// Mitsubishi GX Works2 project: Ex3   PLC: Q03UDV

PROGRAM MAIN
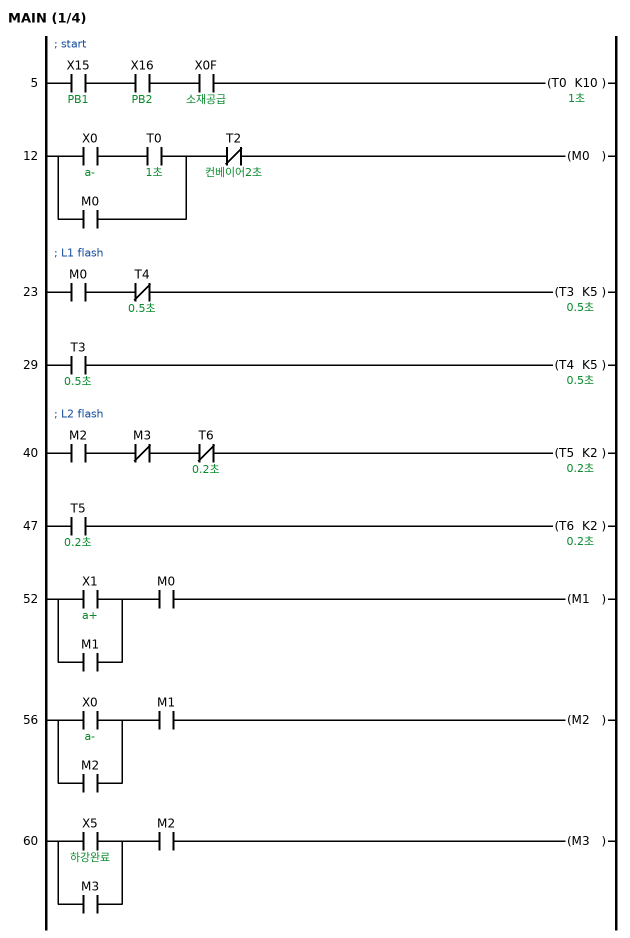
; start
5     LD      X15  ; PB1
      AND     X16  ; PB2
      AND     X0F  ; 소재공급
      OUT     T0 K10  ; 1초
12    LD      X0  ; a-
      AND     T0  ; 1초
      OR      M0
      ANI     T2  ; 컨베이어2초
      OUT     M0
; L1 flash
23    LD      M0
      ANI     T4  ; 0.5초
      OUT     T3 K5  ; 0.5초
29    LD      T3  ; 0.5초
      OUT     T4 K5  ; 0.5초
; L2 flash
40    LD      M2
      ANI     M3
      ANI     T6  ; 0.2초
      OUT     T5 K2  ; 0.2초
47    LD      T5  ; 0.2초
      OUT     T6 K2  ; 0.2초
52    LD      X1  ; a+
      OR      M1
      AND     M0
      OUT     M1
56    LD      X0  ; a-
      OR      M2
      AND     M1
      OUT     M2
60    LD      X5  ; 하강완료
      OR      M3
      AND     M2
      OUT     M3
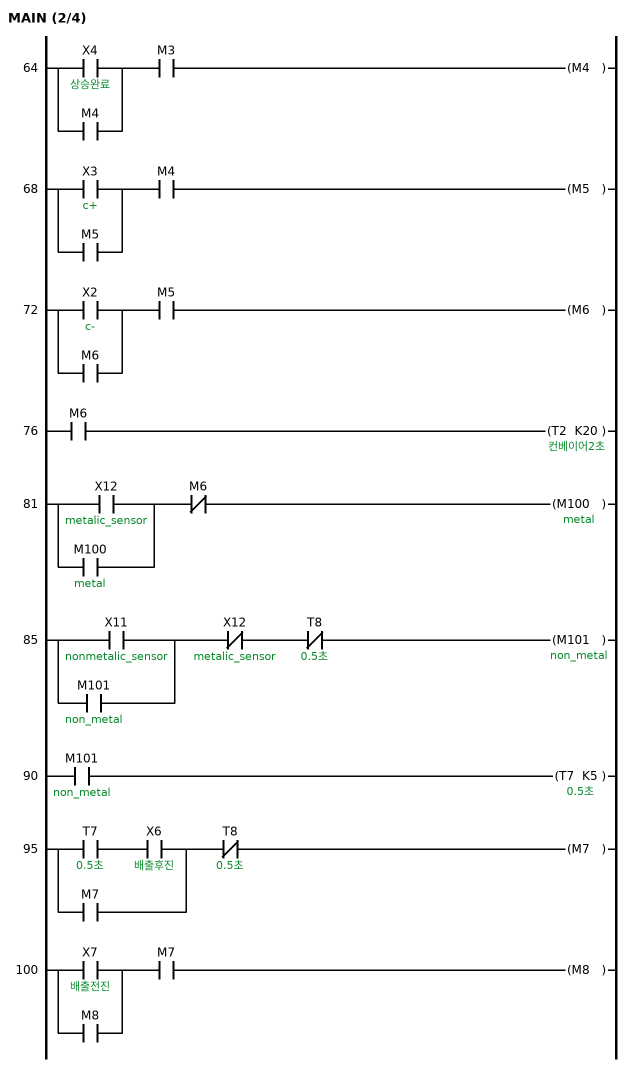
64    LD      X4  ; 상승완료
      OR      M4
      AND     M3
      OUT     M4
68    LD      X3  ; c+
      OR      M5
      AND     M4
      OUT     M5
72    LD      X2  ; c-
      OR      M6
      AND     M5
      OUT     M6
76    LD      M6
      OUT     T2 K20  ; 컨베이어2초
81    LD      X12  ; metalic_sensor
      OR      M100  ; metal
      ANI     M6
      OUT     M100  ; metal
85    LD      X11  ; nonmetalic_sensor
      OR      M101  ; non_metal
      ANI     X12  ; metalic_sensor
      ANI     T8  ; 0.5초
      OUT     M101  ; non_metal
90    LD      M101  ; non_metal
      OUT     T7 K5  ; 0.5초
95    LD      T7  ; 0.5초
      AND     X6  ; 배출후진
      OR      M7
      ANI     T8  ; 0.5초
      OUT     M7
100   LD      X7  ; 배출전진
      OR      M8
      AND     M7
      OUT     M8
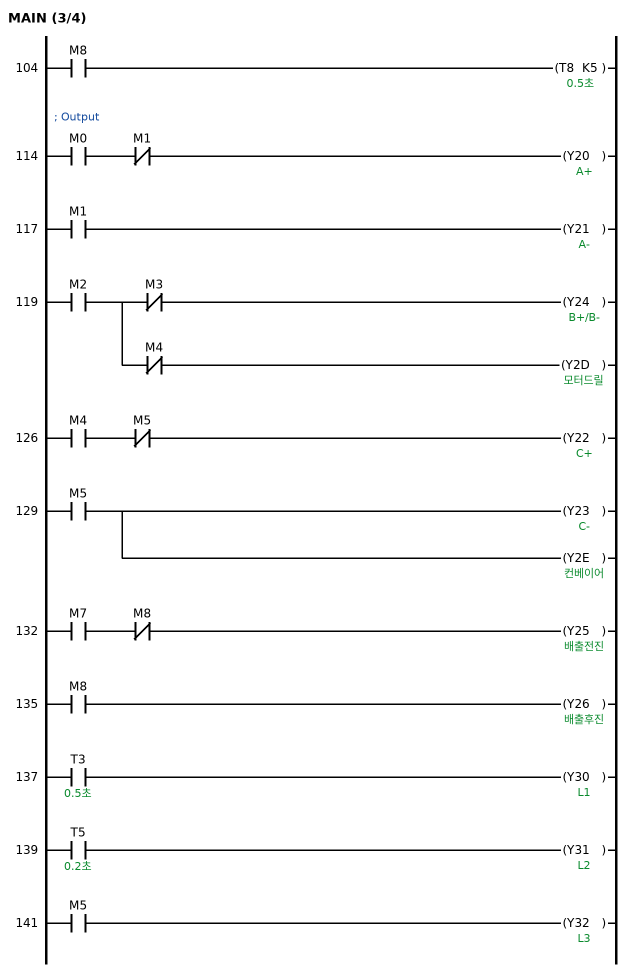
104   LD      M8
      OUT     T8 K5  ; 0.5초
; Output
114   LD      M0
      ANI     M1
      OUT     Y20  ; A+
117   LD      M1
      OUT     Y21  ; A-
119   LD      M2
      MPS
      ANI     M3
      OUT     Y24  ; B+/B-
      MPP
      ANI     M4
      OUT     Y2D  ; 모터드릴
126   LD      M4
      ANI     M5
      OUT     Y22  ; C+
129   LD      M5
      OUT     Y23  ; C-
      OUT     Y2E  ; 컨베이어
132   LD      M7
      ANI     M8
      OUT     Y25  ; 배출전진
135   LD      M8
      OUT     Y26  ; 배출후진
137   LD      T3  ; 0.5초
      OUT     Y30  ; L1
139   LD      T5  ; 0.2초
      OUT     Y31  ; L2
141   LD      M5
      OUT     Y32  ; L3
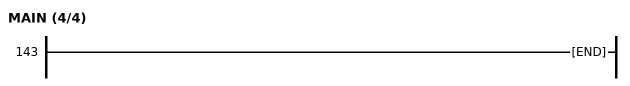
143   END
END_PROGRAM

// device comments not shown above
M102  ; non_metal
